{attribute 'GeneratedUsingTerminal: EP1809-0042-0019'}
{attribute addProperty BoxType "EP1809-0042-0019"}
{attribute addProperty Id "InputAT %I*BOOL1"}
{attribute addProperty CRC "2198356929"}
{attribute addProperty Size "1"}
TYPE DI_X_830843C1 :
STRUCT
	{attribute addProperty Name "Input"}
	Input AT %I* : BOOL;
END_STRUCT
END_TYPE

(* stored: Version 1.2.0.0, ProductVersion 3.1.4024.9
   DUT DI_X_830843C1: Id {5eee5fc5-57ec-40ff-a0f3-e106e8f02f87} *)
